/// Abstract base FB for components
{attribute 'enable_dynamic_creation' := ''}
{attribute 'reflection' := ''}
FUNCTION_BLOCK FB_ComponentBase IMPLEMENTS ITFComponent
VAR
	ii				: INT;
	/// Unique ID of this instance (cam be used as index: P_ComponentPool.aComponents[iID]...)
	iId				: INT;
	/// component type
	eTyp			: E_ComponentType;
	/// component active flag
	bActive			: BOOL;
	/// component state
	eState			: E_ComponentState;
	// Logger
	ILog			: I_Logger;
	/// path of this FB (e.g. for log: P_ComponentPool.fbVirtualMaster)	
    {attribute 'instance-path'} 
    {attribute 'noinit'}
    {attribute 'hide'} 
	sPath			: STRING;
	// object id
	wsObjectId		: WSTRING;

	/// component name
	stName			: ST_Text;
	/// component name
	sBMK			: STRING;
	/// clear text info
	//aSClearText		: ARRAY[0..eLanguage_maxIdx] OF T_MaxString;
	aSClearText		: ST_Text;//T_MaxString;
	
	/// last error debug info
	sLastError		: T_MaxString;
	
	// event handler & source info
	IEvent			: I_EventHandler;
	TcSourceInfo	: FB_TcSourceInfo;
END_VAR

///
/// Abstract base FB for components
/// TP/www.rmth.at/11.2014
///

/// Get's or set's a value indicating whether this component is active or not.
{attribute 'monitoring':='call'}
PROPERTY Active : BOOL
GET
Active := bActive;
END_GET
SET
bActive := Active;
aSClearText := F_CreateDynTextDefaultS(SEL(bActive, 'INACTIVE!', 'ACTIVE!'));
END_SET
END_PROPERTY

METHOD PROTECTED AddLogErr
VAR_INPUT
	sLog : T_MaxString;
END_VAR
// chk
IF ILog = 0 THEN
	RETURN;
END_IF

ILog.AddLog(sLog, WSTRING_TO_STRING(stName.wsName), E_LogLevel.eLogLevel_err);
END_METHOD

METHOD PROTECTED AddLogInf
VAR_INPUT
	sLog : T_MaxString;
END_VAR
// chk
IF ILog = 0 THEN
	RETURN;
END_IF

ILog.AddLog(sLog, WSTRING_TO_STRING(stName.wsName), E_LogLevel.eLogLevel_info);
END_METHOD

METHOD PROTECTED AddLogWrn
VAR_INPUT
	sLog : T_MaxString;
END_VAR
VAR

END_VAR
// chk
IF ILog = 0 THEN
	RETURN;
END_IF

ILog.AddLog(sLog, WSTRING_TO_STRING(stName.wsName), E_LogLevel.eLogLevel_warn);
END_METHOD

{attribute 'monitoring':='call'}
PROPERTY BMK : STRING
GET
BMK := sBMK;
END_GET
SET
sBMK := BMK;
END_SET
END_PROPERTY

/// Get's value representing the component state.
{attribute 'monitoring':='call'}
PROPERTY ClearText : WSTRING(255)
GET
ClearText := aSClearText.wsName;
END_GET
END_PROPERTY

/// Unique component ID (cam be used as index: P_ComponentPool.aComponents[eID]...)
{attribute 'monitoring':='call'}
PROPERTY ID : INT
GET
ID := iId;
END_GET
SET
iId := ID;
END_SET
END_PROPERTY

/// Get's value representing the component state.
{attribute 'monitoring':='call'}
PROPERTY LastError : T_MaxString
GET
LastError := sLastError;
END_GET
END_PROPERTY

PROPERTY Logger : I_Logger
SET
ILog := Logger;
END_SET
END_PROPERTY

METHOD M_InitComponentBase : BOOL
VAR_INPUT
END_VAR
// set up default logger and event handler
ILog := Services.ILog;
IEvent := Services.fbEventHandler;
END_METHOD

METHOD M_InitComponentBaseEx : BOOL
VAR_INPUT
	ILogger			: I_Logger;
	IEventHandler	: I_EventHandler;
END_VAR
ILog := ILogger;
IEvent := IEventHandler;
END_METHOD

PROPERTY Name : ST_Text
GET
Name := stName;
END_GET
SET
stName := Name;
END_SET
END_PROPERTY

PROPERTY PUBLIC NameString : WSTRING(255)
GET
NameString := stName.wsName;
END_GET
END_PROPERTY

PROPERTY ObjectId : WSTRING
GET
ObjectId := wsObjectId;
END_GET
END_PROPERTY

{attribute 'monitoring':='call'}
PROPERTY Path : String
GET
Path := sPath;
END_GET
END_PROPERTY

PROPERTY RefsValid : BOOL
GET
RefsValid := IEvent <> 0;
END_GET
END_PROPERTY

/// Reset component logic
{attribute 'object_name' := 'Reset'}
METHOD Reset
/// abstract base logic reset

sLastError := sEmpty;

// default: set state to ready
eState := E_ComponentState.eComponentState_ready;
END_METHOD

/// Run component logic
{attribute 'object_name' := 'Run'}
METHOD Run : E_ComponentState
VAR
	ii : INT;
END_VAR
/// abstract base logic run

wsObjectId := TO_WSTRING( F_CutInstancePath(sPath) );

// only rdy state may lead to run
IF eState = E_ComponentState.eComponentState_ready THEN
	eState := E_ComponentState.eComponentState_running;
END_IF

Run := eState;
END_METHOD

/// Get's value representing the component state.
{attribute 'monitoring':='call'}
PROPERTY State : E_ComponentState
GET
State := eState;
END_GET
END_PROPERTY

/// Get's value representing the component state.
{attribute 'monitoring':='call'}
PROPERTY StateToString : STRING
GET
CASE eState OF

	eComponentState_none :
		StateToString := 'undefiniert';
	/// Component is resetting
	eComponentState_resetting:
		StateToString := 'wird zurückgesetzt';
	/// Component is ready
	eComponentState_ready:
		StateToString := 'ist bereit';
	/// Component is running
	eComponentState_running:
		StateToString := 'wird ausgeführt';
	/// Component has error
	eComponentState_error:
		StateToString := 'ist fehlerhaft';

END_CASE
END_GET
END_PROPERTY

{attribute 'monitoring':='call'}
PROPERTY Typ : E_ComponentType
GET
Typ := eTyp;
END_GET
END_PROPERTY

END_FUNCTION_BLOCK

(* stored: Version 1.1.0.1
   POU FB_ComponentBase: Id {c18f24bd-a664-4b00-87c6-35388a9e2c13}, SpecialFunc None
   Folder Log: Id {d60d0229-345b-4f21-a527-897b071ec85e}
   Folder Properties: Id {d39cf9c1-a479-4c65-8832-30628ef67dbc}
   Property Active: Id {ad08f73b-d076-4ffc-a47f-109b9002f3f0}
   Get Get: Id {36bc5417-a1df-428f-8558-ccd48ad6e7b2}
   Set Set: Id {91a00653-11d6-478d-b972-77e3e4eb2ccf}
   Method AddLogErr: Id {1fa04579-53a4-4bf7-9485-fed4b63a80f6}
   Method AddLogInf: Id {8f5dc2d6-63af-4a66-8788-1150161b9ec3}
   Method AddLogWrn: Id {c5dba76f-883c-47df-a4a3-7f425d74ab1f}
   Property BMK: Id {3e8ee465-5189-4f2f-9d15-0d6a660f5497}
   Get Get: Id {40debf0c-a597-4287-8751-5255603a498d}
   Set Set: Id {522db787-61e2-4748-b40e-ae4b76e7df74}
   Property ClearText: Id {56ead6a6-eff4-4858-8e9e-da8349489d0c}
   Get Get: Id {b9a876a4-0bf3-4831-bd3b-742033eed1fc}
   Property ID: Id {7adf225e-7442-4f77-874e-8de91565912f}
   Get Get: Id {eb2f488e-56f2-446e-be23-411ca4a9afe8}
   Set Set: Id {41b198fd-6b73-4b90-8815-72b41bb70ddf}
   Property LastError: Id {06cb7fc4-a4a0-4ce5-a61e-ff39359d5455}
   Get Get: Id {ef08fc9c-dbad-4e89-a344-91a0bff8ac28}
   Property Logger: Id {a0145483-d535-4972-887d-7acf62e3e91b}
   Set Set: Id {d2c457c0-a0fd-4903-ad9e-bc9cdf318121}
   Method M_InitComponentBase: Id {08a1113d-250e-48ea-9ee2-595e5c1dfb97}
   Method M_InitComponentBaseEx: Id {d65de655-88e1-4cce-aad2-28b5a41d4593}
   Property Name: Id {97507556-cbd6-4656-a4b4-7ef03ea2ff1e}
   Get Get: Id {0e45fe35-49fc-47f1-97fe-c7f0eb7a6261}
   Set Set: Id {46008dd6-890e-4fe4-a735-05ed8de2d0f7}
   Property NameString: Id {dd0a9030-a1e1-4242-b530-80defac285f6}
   Get Get: Id {1b227500-9a9a-4849-b566-94665e2acf34}
   Property ObjectId: Id {6151cd1a-ec0a-4780-962a-396a138c611b}
   Get Get: Id {99d3fba7-71a7-4d81-9b75-f46e5870f58d}
   Property Path: Id {f15c3da9-69b6-42be-b750-91438e4fc191}
   Get Get: Id {54b2c794-d6e0-472b-8241-5b86ba340b29}
   Property RefsValid: Id {89a3ca2b-9a2f-4d2d-a33a-74f607804482}
   Get Get: Id {a66b32cb-c14f-48dc-873e-71a5d161ca8b}
   Method Reset: Id {7800391a-478c-4265-bd45-1c25f898c8f4}
   Method Run: Id {04530f9f-040a-4517-8bda-6e0d48f73e41}
   Property State: Id {d68fb6ae-0af8-44c3-bb4d-32b1388481b9}
   Get Get: Id {f34831ab-8558-4954-8527-8fd474b2d71e}
   Property StateToString: Id {bffb55f1-1ef3-4369-ab66-e92ce785efbd}
   Get Get: Id {a3e43248-1732-4fcc-9614-52c3ff99ce09}
   Property Typ: Id {987dd2cf-7ace-4cc4-856e-8b41f907e2c3}
   Get Get: Id {4aca47e7-510b-43f6-9b4f-e58faabf961a} *)
